FUNCTION_BLOCK InputDecompressor (* Basic Function Block Type *)
  (* Standard: 61499-2 *)
  (* Version 0.0, 11/1/2016, Dmitry, nxtControl GmbH, Template *)
  PACKAGE Main;
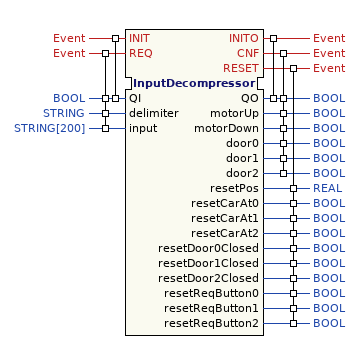
  EVENT_INPUT
    INIT WITH QI; (* Initialization Request *)
    REQ WITH QI, delimiter, input; (* Normal Execution Request *)
  END_EVENT
  EVENT_OUTPUT
    INITO WITH QO; (* Initialization Confirm *)
    CNF WITH QO, motorUp, motorDown, door0, door1, door2; (* Execution Confirmation *)
    RESET WITH resetPos, resetCarAt0, resetCarAt1, resetCarAt2, resetDoor0Closed, resetDoor1Closed, resetDoor2Closed, resetReqButton0, resetReqButton1, resetReqButton2;
  END_EVENT
  VAR_INPUT
    QI : BOOL; (* Input event qualifier *)
    delimiter : STRING;
    input : STRING[200];
  END_VAR
  VAR_OUTPUT
    QO : BOOL; (* Output event qualifier *)
    motorUp : BOOL;
    motorDown : BOOL;
    door0 : BOOL;
    door1 : BOOL;
    door2 : BOOL;
    resetPos : REAL;
    resetCarAt0 : BOOL;
    resetCarAt1 : BOOL;
    resetCarAt2 : BOOL;
    resetDoor0Closed : BOOL;
    resetDoor1Closed : BOOL;
    resetDoor2Closed : BOOL;
    resetReqButton0 : BOOL;
    resetReqButton1 : BOOL;
    resetReqButton2 : BOOL;
  END_VAR
  VAR
    reset : BOOL;
    subs : ARRAY [0..13] OF STRING;
  END_VAR
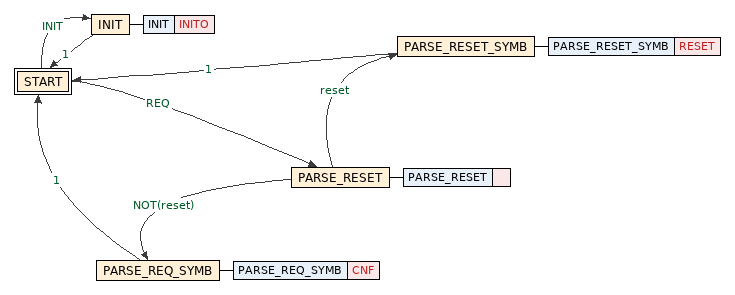
  EC_STATES
    START; (* Initial State *)
    INIT : INIT -> INITO; (* Initialization *)
    PARSE_REQ_SYMB : PARSE_REQ_SYMB -> CNF;
    PARSE_RESET_SYMB : PARSE_RESET_SYMB -> RESET;
    PARSE_RESET : PARSE_RESET;
  END_STATES
  EC_TRANSITIONS
    START TO INIT := INIT;
    INIT TO START := 1;
    START TO PARSE_RESET := REQ;
    PARSE_RESET TO PARSE_RESET_SYMB := reset;
    PARSE_RESET TO PARSE_REQ_SYMB := NOT(reset);
    PARSE_REQ_SYMB TO START := 1;
    PARSE_RESET_SYMB TO START := 1;
  END_TRANSITIONS
  ALGORITHM INIT IN ST: (* Initialization algorithm *)
QO := TRUE;
  END_ALGORITHM
  ALGORITHM REQ IN ST: (* Normally executed algorithm *)
;
  END_ALGORITHM
  ALGORITHM PARSE_RESET IN ST:
VAR
	i: INT;
END_VAR;
i := 1;
(*WHILE MID(input, 1, i) <> delimiter DO
	i := i + 1;
END_WHILE;*)
reset := STRING_TO_BOOL(MID(input, i, 1));
  END_ALGORITHM
  ALGORITHM PARSE_RESET_SYMB IN ST:
VAR
	length: INT;
	i : INT;
	prev: INT;
	substr : ARRAY[1..11] OF STRING;
	num : INT;
	cur: INT;
END_VAR;
length := DINT_TO_INT(LEN(input));
prev := 1;
cur := 1;
FOR i := 1 TO length DO
	IF (MID(input,1,i) = delimiter) THEN

		substr[cur] := MID(input, i - prev, prev);//input.DATA[prev, i-1];
		cur := cur + 1;
		prev := i + 1;
	END_IF;
END_FOR;

(*resetButtonFloor0 := STRING_TO_BOOL(subs[1]);
resetButtonFloor1 := STRING_TO_BOOL(subs[2]);
resetButtonFloor2 := STRING_TO_BOOL(subs[3]);*)

resetReqButton0 := STRING_TO_BOOL(substr[2]);
resetReqButton1 := STRING_TO_BOOL(substr[3]);
resetReqButton2 := STRING_TO_BOOL(substr[4]);

resetCarAt0 := STRING_TO_BOOL(substr[5]);
resetCarAt1 := STRING_TO_BOOL(substr[6]);
resetCarAt2 := STRING_TO_BOOL(substr[7]);

resetDoor0Closed := STRING_TO_BOOL(substr[8]);
resetDoor1Closed := STRING_TO_BOOL(substr[9]);
resetDoor2Closed := STRING_TO_BOOL(substr[10]);

resetPos := STRING_TO_REAL(substr[11]);
  END_ALGORITHM
  ALGORITHM PARSE_REQ_SYMB IN ST:
VAR
	length: INT;
	i : INT;
	prev: INT;
	substr : ARRAY[1..6] OF STRING;
	num : INT;
	cur: INT;
END_VAR;
length := DINT_TO_INT(LEN(input));
prev := 1;
cur := 1;
FOR i := 1 TO length DO
	IF (MID(input,1,i) = delimiter) THEN
		substr[cur] := MID(input, i - prev, prev);//input.DATA[prev, i-1];
		cur := cur + 1;
		prev := i + 1;
	END_IF;
END_FOR;
motorUp := STRING_TO_BOOL(substr[2]);
motorDown := STRING_TO_BOOL(substr[3]);
door0 := STRING_TO_BOOL(substr[4]);
door1 := STRING_TO_BOOL(substr[5]);
door2 := STRING_TO_BOOL(substr[6]);
(*requestFloor0 := STRING_TO_BOOL(substr[7]);
requestFloor1 := STRING_TO_BOOL(substr[8]);
requestFloor2 := STRING_TO_BOOL(substr[9]);*)
  END_ALGORITHM
END_FUNCTION_BLOCK
